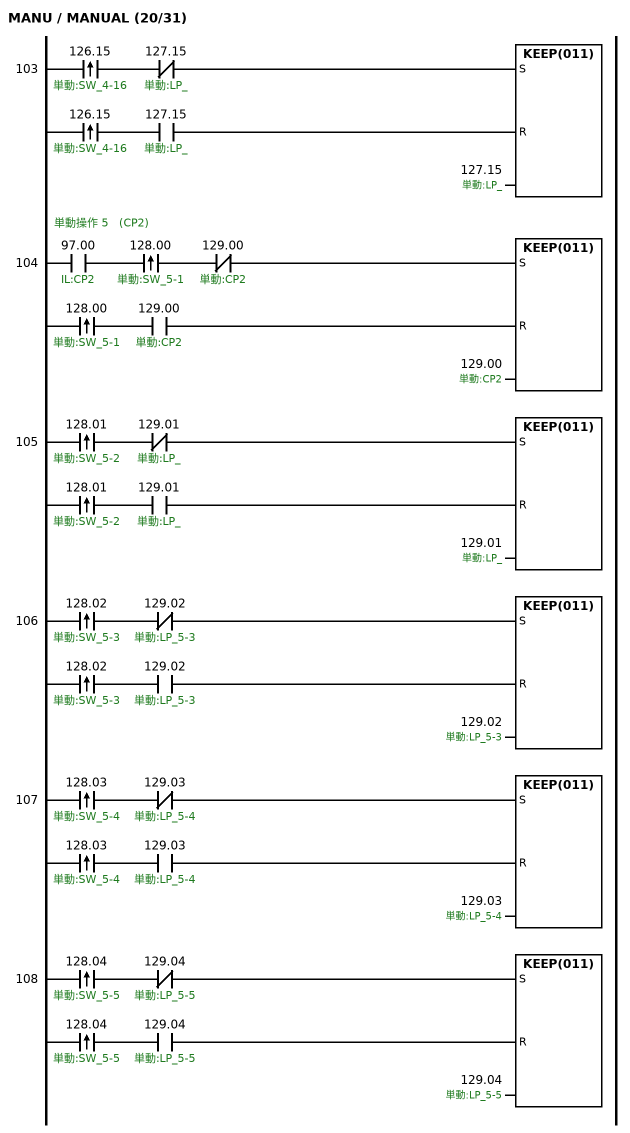
; [picture p72: MANU / MANUAL, rungs 103-108]
; rung 103
@LD 126.15  ; 単動:SW_4-16
ANDNOT 127.15  ; 単動:LP_
@LD 126.15  ; 単動:SW_4-16
AND 127.15  ; 単動:LP_
KEEP(011) 127.15  ; 単動:LP_
; rung 104: 単動操作 5   (CP2)
LD 97.00  ; IL:CP2
@AND 128.00  ; 単動:SW_5-1
ANDNOT 129.00  ; 単動:CP2
@LD 128.00  ; 単動:SW_5-1
AND 129.00  ; 単動:CP2
KEEP(011) 129.00  ; 単動:CP2
; rung 105
@LD 128.01  ; 単動:SW_5-2
ANDNOT 129.01  ; 単動:LP_
@LD 128.01  ; 単動:SW_5-2
AND 129.01  ; 単動:LP_
KEEP(011) 129.01  ; 単動:LP_
; rung 106
@LD 128.02  ; 単動:SW_5-3
ANDNOT 129.02  ; 単動:LP_5-3
@LD 128.02  ; 単動:SW_5-3
AND 129.02  ; 単動:LP_5-3
KEEP(011) 129.02  ; 単動:LP_5-3
; rung 107
@LD 128.03  ; 単動:SW_5-4
ANDNOT 129.03  ; 単動:LP_5-4
@LD 128.03  ; 単動:SW_5-4
AND 129.03  ; 単動:LP_5-4
KEEP(011) 129.03  ; 単動:LP_5-4
; rung 108
@LD 128.04  ; 単動:SW_5-5
ANDNOT 129.04  ; 単動:LP_5-5
@LD 128.04  ; 単動:SW_5-5
AND 129.04  ; 単動:LP_5-5
KEEP(011) 129.04  ; 単動:LP_5-5

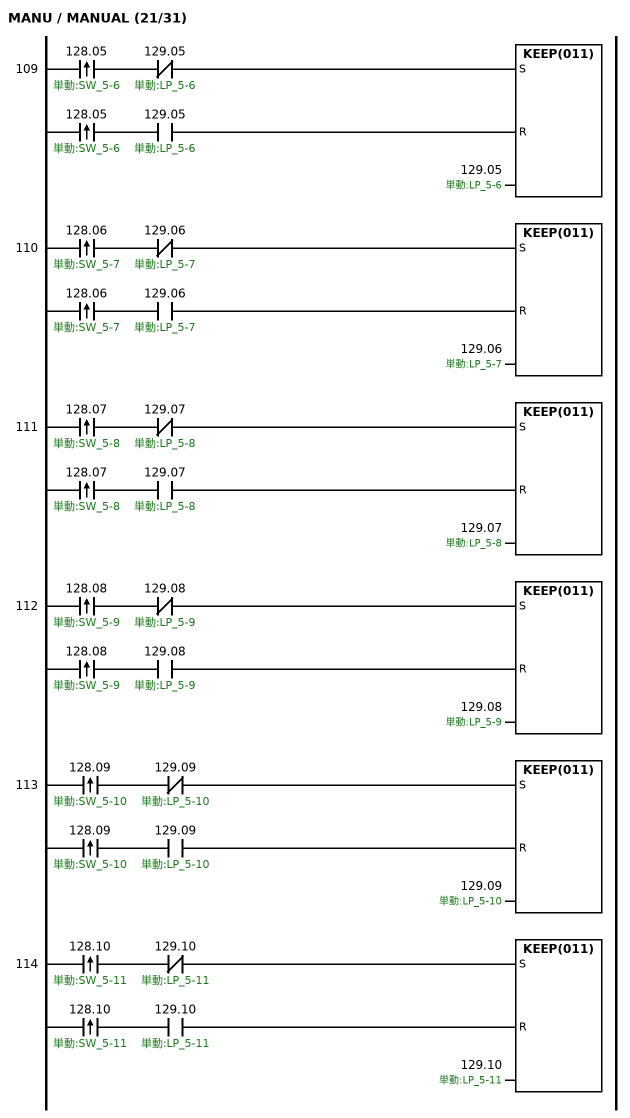
; rung 109
@LD 128.05  ; 単動:SW_5-6
ANDNOT 129.05  ; 単動:LP_5-6
@LD 128.05  ; 単動:SW_5-6
AND 129.05  ; 単動:LP_5-6
KEEP(011) 129.05  ; 単動:LP_5-6
; rung 110
@LD 128.06  ; 単動:SW_5-7
ANDNOT 129.06  ; 単動:LP_5-7
@LD 128.06  ; 単動:SW_5-7
AND 129.06  ; 単動:LP_5-7
KEEP(011) 129.06  ; 単動:LP_5-7
; rung 111
@LD 128.07  ; 単動:SW_5-8
ANDNOT 129.07  ; 単動:LP_5-8
@LD 128.07  ; 単動:SW_5-8
AND 129.07  ; 単動:LP_5-8
KEEP(011) 129.07  ; 単動:LP_5-8
; rung 112
@LD 128.08  ; 単動:SW_5-9
ANDNOT 129.08  ; 単動:LP_5-9
@LD 128.08  ; 単動:SW_5-9
AND 129.08  ; 単動:LP_5-9
KEEP(011) 129.08  ; 単動:LP_5-9
; rung 113
@LD 128.09  ; 単動:SW_5-10
ANDNOT 129.09  ; 単動:LP_5-10
@LD 128.09  ; 単動:SW_5-10
AND 129.09  ; 単動:LP_5-10
KEEP(011) 129.09  ; 単動:LP_5-10
; rung 114
@LD 128.10  ; 単動:SW_5-11
ANDNOT 129.10  ; 単動:LP_5-11
@LD 128.10  ; 単動:SW_5-11
AND 129.10  ; 単動:LP_5-11
KEEP(011) 129.10  ; 単動:LP_5-11

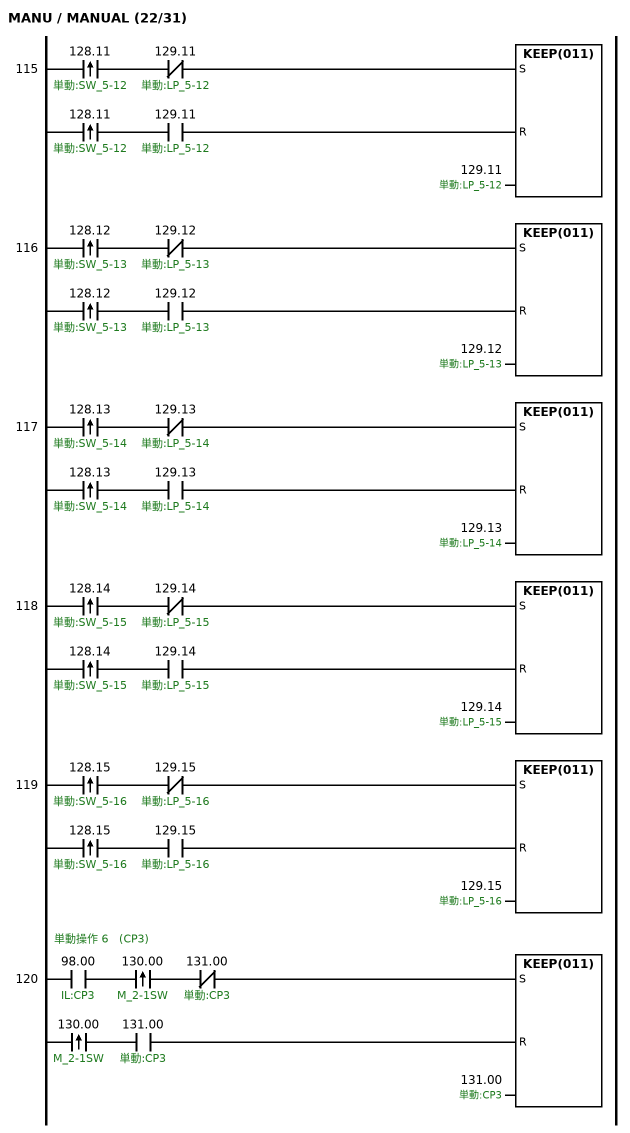
; rung 115
@LD 128.11  ; 単動:SW_5-12
ANDNOT 129.11  ; 単動:LP_5-12
@LD 128.11  ; 単動:SW_5-12
AND 129.11  ; 単動:LP_5-12
KEEP(011) 129.11  ; 単動:LP_5-12
; rung 116
@LD 128.12  ; 単動:SW_5-13
ANDNOT 129.12  ; 単動:LP_5-13
@LD 128.12  ; 単動:SW_5-13
AND 129.12  ; 単動:LP_5-13
KEEP(011) 129.12  ; 単動:LP_5-13
; rung 117
@LD 128.13  ; 単動:SW_5-14
ANDNOT 129.13  ; 単動:LP_5-14
@LD 128.13  ; 単動:SW_5-14
AND 129.13  ; 単動:LP_5-14
KEEP(011) 129.13  ; 単動:LP_5-14
; rung 118
@LD 128.14  ; 単動:SW_5-15
ANDNOT 129.14  ; 単動:LP_5-15
@LD 128.14  ; 単動:SW_5-15
AND 129.14  ; 単動:LP_5-15
KEEP(011) 129.14  ; 単動:LP_5-15
; rung 119
@LD 128.15  ; 単動:SW_5-16
ANDNOT 129.15  ; 単動:LP_5-16
@LD 128.15  ; 単動:SW_5-16
AND 129.15  ; 単動:LP_5-16
KEEP(011) 129.15  ; 単動:LP_5-16
; rung 120: 単動操作 6   (CP3)
LD 98.00  ; IL:CP3
@AND 130.00  ; M_2-1SW
ANDNOT 131.00  ; 単動:CP3
@LD 130.00  ; M_2-1SW
AND 131.00  ; 単動:CP3
KEEP(011) 131.00  ; 単動:CP3

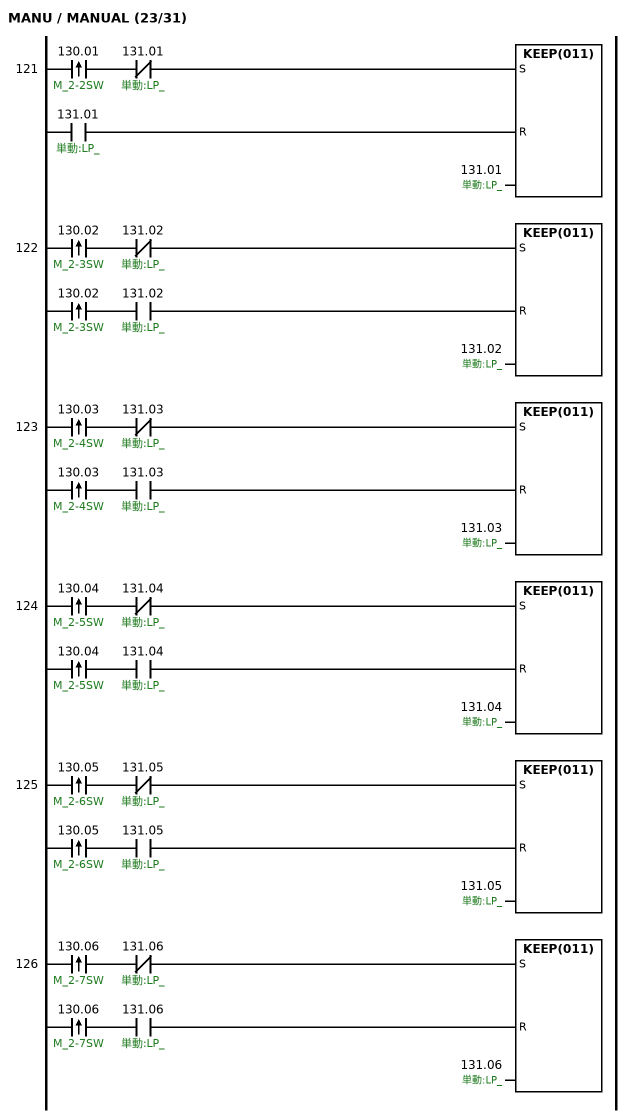
; rung 121
@LD 130.01  ; M_2-2SW
ANDNOT 131.01  ; 単動:LP_
LD 131.01  ; 単動:LP_
KEEP(011) 131.01  ; 単動:LP_
; rung 122
@LD 130.02  ; M_2-3SW
ANDNOT 131.02  ; 単動:LP_
@LD 130.02  ; M_2-3SW
AND 131.02  ; 単動:LP_
KEEP(011) 131.02  ; 単動:LP_
; rung 123
@LD 130.03  ; M_2-4SW
ANDNOT 131.03  ; 単動:LP_
@LD 130.03  ; M_2-4SW
AND 131.03  ; 単動:LP_
KEEP(011) 131.03  ; 単動:LP_
; rung 124
@LD 130.04  ; M_2-5SW
ANDNOT 131.04  ; 単動:LP_
@LD 130.04  ; M_2-5SW
AND 131.04  ; 単動:LP_
KEEP(011) 131.04  ; 単動:LP_
; rung 125
@LD 130.05  ; M_2-6SW
ANDNOT 131.05  ; 単動:LP_
@LD 130.05  ; M_2-6SW
AND 131.05  ; 単動:LP_
KEEP(011) 131.05  ; 単動:LP_
; rung 126
@LD 130.06  ; M_2-7SW
ANDNOT 131.06  ; 単動:LP_
@LD 130.06  ; M_2-7SW
AND 131.06  ; 単動:LP_
KEEP(011) 131.06  ; 単動:LP_

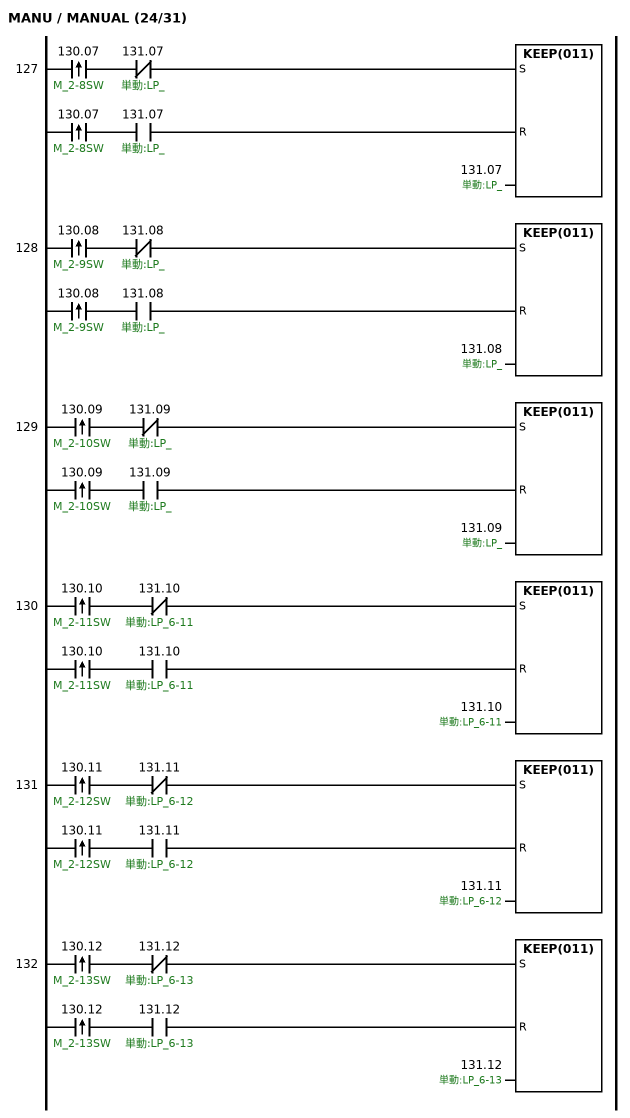
; rung 127
@LD 130.07  ; M_2-8SW
ANDNOT 131.07  ; 単動:LP_
@LD 130.07  ; M_2-8SW
AND 131.07  ; 単動:LP_
KEEP(011) 131.07  ; 単動:LP_
; rung 128
@LD 130.08  ; M_2-9SW
ANDNOT 131.08  ; 単動:LP_
@LD 130.08  ; M_2-9SW
AND 131.08  ; 単動:LP_
KEEP(011) 131.08  ; 単動:LP_
; rung 129
@LD 130.09  ; M_2-10SW
ANDNOT 131.09  ; 単動:LP_
@LD 130.09  ; M_2-10SW
AND 131.09  ; 単動:LP_
KEEP(011) 131.09  ; 単動:LP_
; rung 130
@LD 130.10  ; M_2-11SW
ANDNOT 131.10  ; 単動:LP_6-11
@LD 130.10  ; M_2-11SW
AND 131.10  ; 単動:LP_6-11
KEEP(011) 131.10  ; 単動:LP_6-11
; rung 131
@LD 130.11  ; M_2-12SW
ANDNOT 131.11  ; 単動:LP_6-12
@LD 130.11  ; M_2-12SW
AND 131.11  ; 単動:LP_6-12
KEEP(011) 131.11  ; 単動:LP_6-12
; rung 132
@LD 130.12  ; M_2-13SW
ANDNOT 131.12  ; 単動:LP_6-13
@LD 130.12  ; M_2-13SW
AND 131.12  ; 単動:LP_6-13
KEEP(011) 131.12  ; 単動:LP_6-13

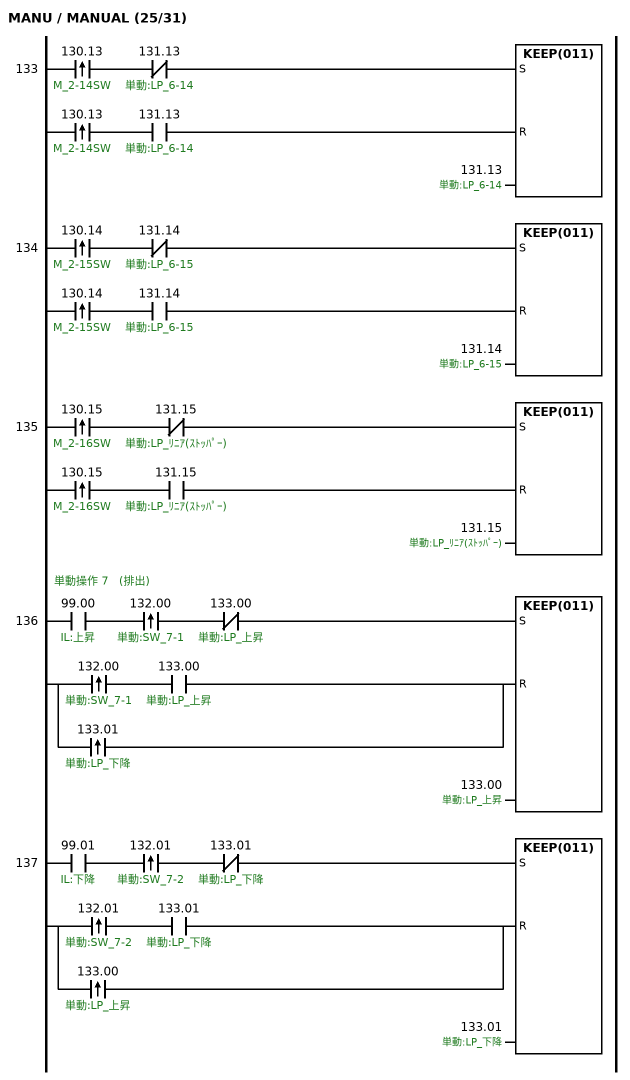
; rung 133
@LD 130.13  ; M_2-14SW
ANDNOT 131.13  ; 単動:LP_6-14
@LD 130.13  ; M_2-14SW
AND 131.13  ; 単動:LP_6-14
KEEP(011) 131.13  ; 単動:LP_6-14
; rung 134
@LD 130.14  ; M_2-15SW
ANDNOT 131.14  ; 単動:LP_6-15
@LD 130.14  ; M_2-15SW
AND 131.14  ; 単動:LP_6-15
KEEP(011) 131.14  ; 単動:LP_6-15
; rung 135
@LD 130.15  ; M_2-16SW
ANDNOT 131.15  ; 単動:LP_ﾘﾆｱ(ｽﾄｯﾊﾟｰ)
@LD 130.15  ; M_2-16SW
AND 131.15  ; 単動:LP_ﾘﾆｱ(ｽﾄｯﾊﾟｰ)
KEEP(011) 131.15  ; 単動:LP_ﾘﾆｱ(ｽﾄｯﾊﾟｰ)
; rung 136: 単動操作 7   (排出)
LD 99.00  ; IL:上昇
@AND 132.00  ; 単動:SW_7-1
ANDNOT 133.00  ; 単動:LP_上昇
@LD 132.00  ; 単動:SW_7-1
AND 133.00  ; 単動:LP_上昇
@OR 133.01  ; 単動:LP_下降
KEEP(011) 133.00  ; 単動:LP_上昇
; rung 137
LD 99.01  ; IL:下降
@AND 132.01  ; 単動:SW_7-2
ANDNOT 133.01  ; 単動:LP_下降
@LD 132.01  ; 単動:SW_7-2
AND 133.01  ; 単動:LP_下降
@OR 133.00  ; 単動:LP_上昇
KEEP(011) 133.01  ; 単動:LP_下降

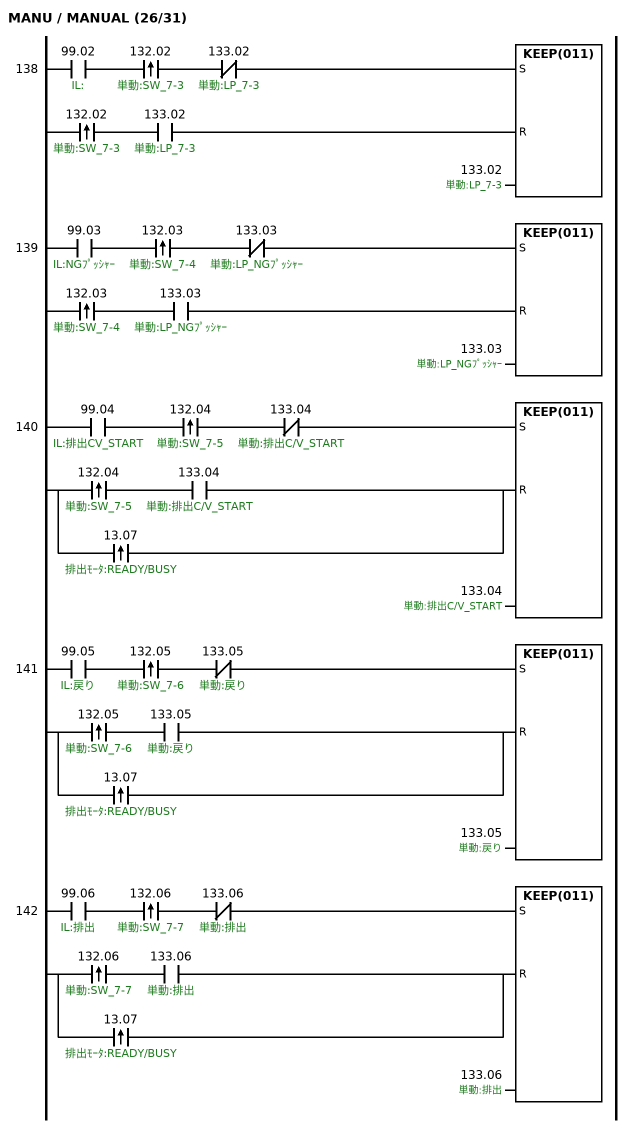
; rung 138
LD 99.02  ; IL:
@AND 132.02  ; 単動:SW_7-3
ANDNOT 133.02  ; 単動:LP_7-3
@LD 132.02  ; 単動:SW_7-3
AND 133.02  ; 単動:LP_7-3
KEEP(011) 133.02  ; 単動:LP_7-3
; rung 139
LD 99.03  ; IL:NGﾌﾟｯｼｬｰ
@AND 132.03  ; 単動:SW_7-4
ANDNOT 133.03  ; 単動:LP_NGﾌﾟｯｼｬｰ
@LD 132.03  ; 単動:SW_7-4
AND 133.03  ; 単動:LP_NGﾌﾟｯｼｬｰ
KEEP(011) 133.03  ; 単動:LP_NGﾌﾟｯｼｬｰ
; rung 140
LD 99.04  ; IL:排出CV_START
@AND 132.04  ; 単動:SW_7-5
ANDNOT 133.04  ; 単動:排出C/V_START
@LD 132.04  ; 単動:SW_7-5
AND 133.04  ; 単動:排出C/V_START
@OR 13.07  ; 排出ﾓｰﾀ:READY/BUSY
KEEP(011) 133.04  ; 単動:排出C/V_START
; rung 141
LD 99.05  ; IL:戻り
@AND 132.05  ; 単動:SW_7-6
ANDNOT 133.05  ; 単動:戻り
@LD 132.05  ; 単動:SW_7-6
AND 133.05  ; 単動:戻り
@OR 13.07  ; 排出ﾓｰﾀ:READY/BUSY
KEEP(011) 133.05  ; 単動:戻り
; rung 142
LD 99.06  ; IL:排出
@AND 132.06  ; 単動:SW_7-7
ANDNOT 133.06  ; 単動:排出
@LD 132.06  ; 単動:SW_7-7
AND 133.06  ; 単動:排出
@OR 13.07  ; 排出ﾓｰﾀ:READY/BUSY
KEEP(011) 133.06  ; 単動:排出

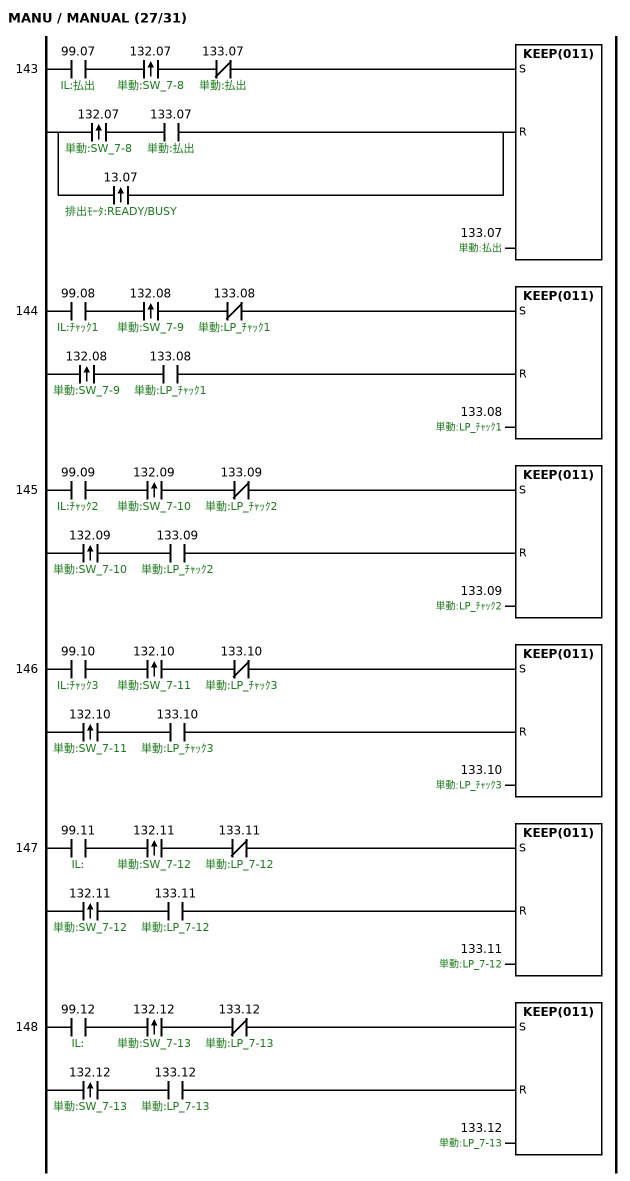
; rung 143
LD 99.07  ; IL:払出
@AND 132.07  ; 単動:SW_7-8
ANDNOT 133.07  ; 単動:払出
@LD 132.07  ; 単動:SW_7-8
AND 133.07  ; 単動:払出
@OR 13.07  ; 排出ﾓｰﾀ:READY/BUSY
KEEP(011) 133.07  ; 単動:払出
; rung 144
LD 99.08  ; IL:ﾁｬｯｸ1
@AND 132.08  ; 単動:SW_7-9
ANDNOT 133.08  ; 単動:LP_ﾁｬｯｸ1
@LD 132.08  ; 単動:SW_7-9
AND 133.08  ; 単動:LP_ﾁｬｯｸ1
KEEP(011) 133.08  ; 単動:LP_ﾁｬｯｸ1
; rung 145
LD 99.09  ; IL:ﾁｬｯｸ2
@AND 132.09  ; 単動:SW_7-10
ANDNOT 133.09  ; 単動:LP_ﾁｬｯｸ2
@LD 132.09  ; 単動:SW_7-10
AND 133.09  ; 単動:LP_ﾁｬｯｸ2
KEEP(011) 133.09  ; 単動:LP_ﾁｬｯｸ2
; rung 146
LD 99.10  ; IL:ﾁｬｯｸ3
@AND 132.10  ; 単動:SW_7-11
ANDNOT 133.10  ; 単動:LP_ﾁｬｯｸ3
@LD 132.10  ; 単動:SW_7-11
AND 133.10  ; 単動:LP_ﾁｬｯｸ3
KEEP(011) 133.10  ; 単動:LP_ﾁｬｯｸ3
; rung 147
LD 99.11  ; IL:
@AND 132.11  ; 単動:SW_7-12
ANDNOT 133.11  ; 単動:LP_7-12
@LD 132.11  ; 単動:SW_7-12
AND 133.11  ; 単動:LP_7-12
KEEP(011) 133.11  ; 単動:LP_7-12
; rung 148
LD 99.12  ; IL:
@AND 132.12  ; 単動:SW_7-13
ANDNOT 133.12  ; 単動:LP_7-13
@LD 132.12  ; 単動:SW_7-13
AND 133.12  ; 単動:LP_7-13
KEEP(011) 133.12  ; 単動:LP_7-13

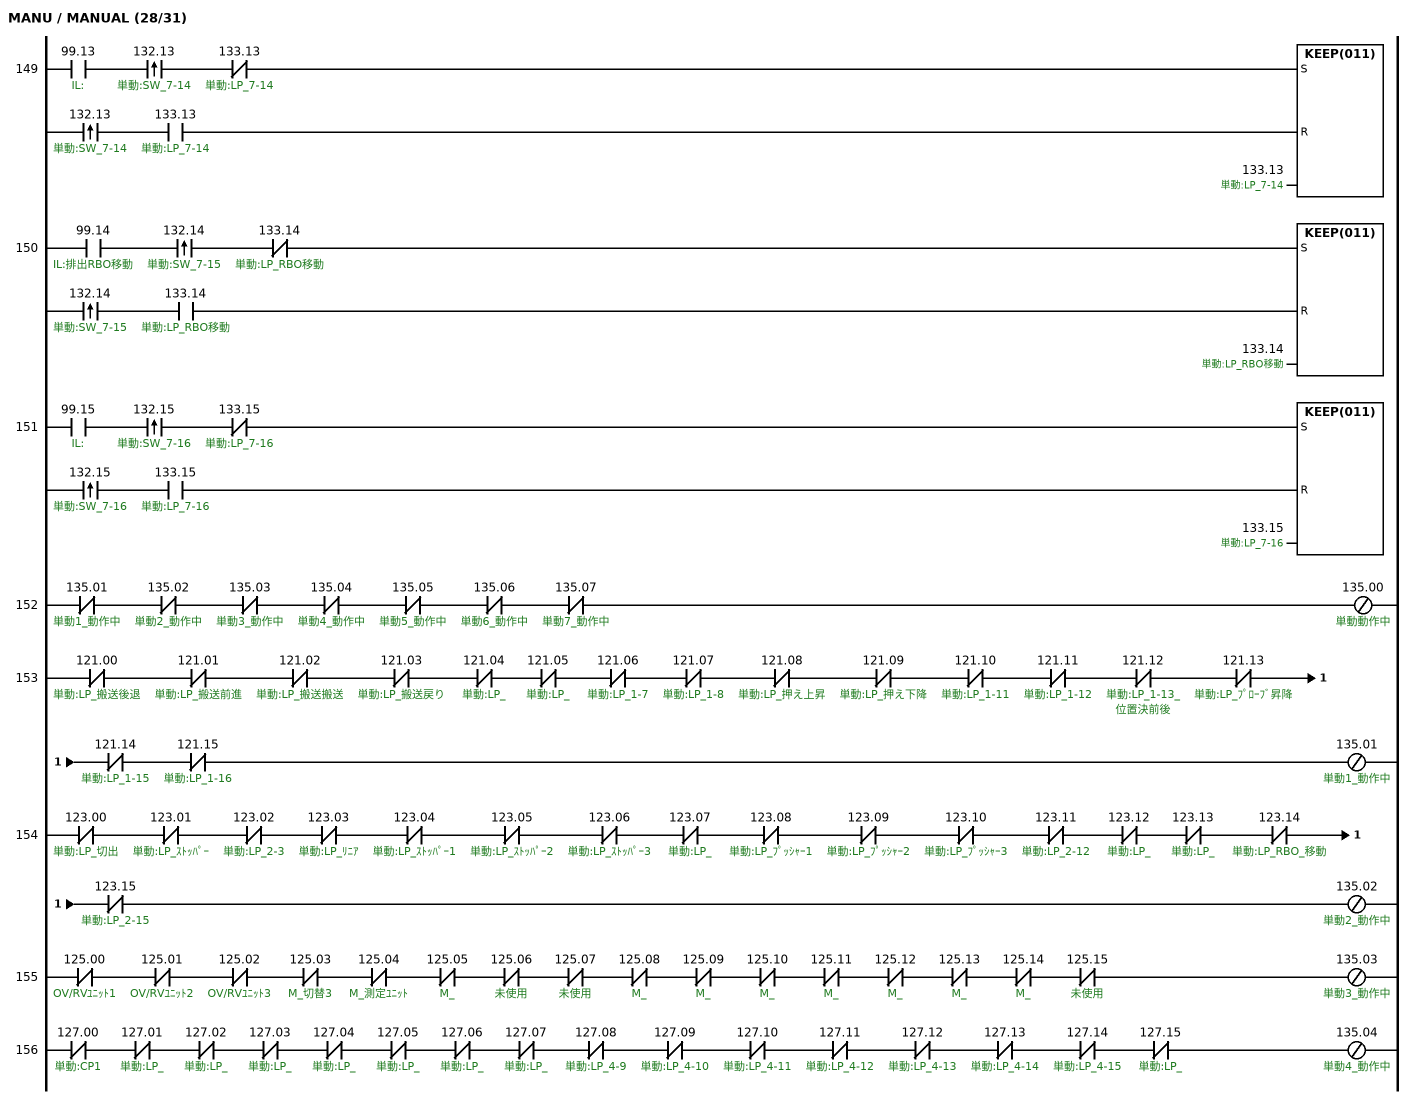
; rung 149
LD 99.13  ; IL:
@AND 132.13  ; 単動:SW_7-14
ANDNOT 133.13  ; 単動:LP_7-14
@LD 132.13  ; 単動:SW_7-14
AND 133.13  ; 単動:LP_7-14
KEEP(011) 133.13  ; 単動:LP_7-14
; rung 150
LD 99.14  ; IL:排出RBO移動
@AND 132.14  ; 単動:SW_7-15
ANDNOT 133.14  ; 単動:LP_RBO移動
@LD 132.14  ; 単動:SW_7-15
AND 133.14  ; 単動:LP_RBO移動
KEEP(011) 133.14  ; 単動:LP_RBO移動
; rung 151
LD 99.15  ; IL:
@AND 132.15  ; 単動:SW_7-16
ANDNOT 133.15  ; 単動:LP_7-16
@LD 132.15  ; 単動:SW_7-16
AND 133.15  ; 単動:LP_7-16
KEEP(011) 133.15  ; 単動:LP_7-16
; rung 152
LDNOT 135.01  ; 単動1_動作中
ANDNOT 135.02  ; 単動2_動作中
ANDNOT 135.03  ; 単動3_動作中
ANDNOT 135.04  ; 単動4_動作中
ANDNOT 135.05  ; 単動5_動作中
ANDNOT 135.06  ; 単動6_動作中
ANDNOT 135.07  ; 単動7_動作中
OUTNOT 135.00  ; 単動動作中
; rung 153
LDNOT 121.00  ; 単動:LP_搬送後退
ANDNOT 121.01  ; 単動:LP_搬送前進
ANDNOT 121.02  ; 単動:LP_搬送搬送
ANDNOT 121.03  ; 単動:LP_搬送戻り
ANDNOT 121.04  ; 単動:LP_
ANDNOT 121.05  ; 単動:LP_
ANDNOT 121.06  ; 単動:LP_1-7
ANDNOT 121.07  ; 単動:LP_1-8
ANDNOT 121.08  ; 単動:LP_押え上昇
ANDNOT 121.09  ; 単動:LP_押え下降
ANDNOT 121.10  ; 単動:LP_1-11
ANDNOT 121.11  ; 単動:LP_1-12
ANDNOT 121.12  ; 単動:LP_1-13_位置決前後
ANDNOT 121.13  ; 単動:LP_ﾌﾟﾛｰﾌﾞ昇降
ANDNOT 121.14  ; 単動:LP_1-15
ANDNOT 121.15  ; 単動:LP_1-16
OUTNOT 135.01  ; 単動1_動作中
; rung 154
LDNOT 123.00  ; 単動:LP_切出
ANDNOT 123.01  ; 単動:LP_ｽﾄｯﾊﾟｰ
ANDNOT 123.02  ; 単動:LP_2-3
ANDNOT 123.03  ; 単動:LP_ﾘﾆｱ
ANDNOT 123.04  ; 単動:LP_ｽﾄｯﾊﾟｰ1
ANDNOT 123.05  ; 単動:LP_ｽﾄｯﾊﾟｰ2
ANDNOT 123.06  ; 単動:LP_ｽﾄｯﾊﾟｰ3
ANDNOT 123.07  ; 単動:LP_
ANDNOT 123.08  ; 単動:LP_ﾌﾟｯｼｬｰ1
ANDNOT 123.09  ; 単動:LP_ﾌﾟｯｼｬｰ2
ANDNOT 123.10  ; 単動:LP_ﾌﾟｯｼｬｰ3
ANDNOT 123.11  ; 単動:LP_2-12
ANDNOT 123.12  ; 単動:LP_
ANDNOT 123.13  ; 単動:LP_
ANDNOT 123.14  ; 単動:LP_RBO_移動
ANDNOT 123.15  ; 単動:LP_2-15
OUTNOT 135.02  ; 単動2_動作中
; rung 155
LDNOT 125.00  ; OV/RVﾕﾆｯﾄ1
ANDNOT 125.01  ; OV/RVﾕﾆｯﾄ2
ANDNOT 125.02  ; OV/RVﾕﾆｯﾄ3
ANDNOT 125.03  ; M_切替3
ANDNOT 125.04  ; M_測定ﾕﾆｯﾄ
ANDNOT 125.05  ; M_
ANDNOT 125.06  ; 未使用
ANDNOT 125.07  ; 未使用
ANDNOT 125.08  ; M_
ANDNOT 125.09  ; M_
ANDNOT 125.10  ; M_
ANDNOT 125.11  ; M_
ANDNOT 125.12  ; M_
ANDNOT 125.13  ; M_
ANDNOT 125.14  ; M_
ANDNOT 125.15  ; 未使用
OUTNOT 135.03  ; 単動3_動作中
; rung 156
LDNOT 127.00  ; 単動:CP1
ANDNOT 127.01  ; 単動:LP_
ANDNOT 127.02  ; 単動:LP_
ANDNOT 127.03  ; 単動:LP_
ANDNOT 127.04  ; 単動:LP_
ANDNOT 127.05  ; 単動:LP_
ANDNOT 127.06  ; 単動:LP_
ANDNOT 127.07  ; 単動:LP_
ANDNOT 127.08  ; 単動:LP_4-9
ANDNOT 127.09  ; 単動:LP_4-10
ANDNOT 127.10  ; 単動:LP_4-11
ANDNOT 127.11  ; 単動:LP_4-12
ANDNOT 127.12  ; 単動:LP_4-13
ANDNOT 127.13  ; 単動:LP_4-14
ANDNOT 127.14  ; 単動:LP_4-15
ANDNOT 127.15  ; 単動:LP_
OUTNOT 135.04  ; 単動4_動作中

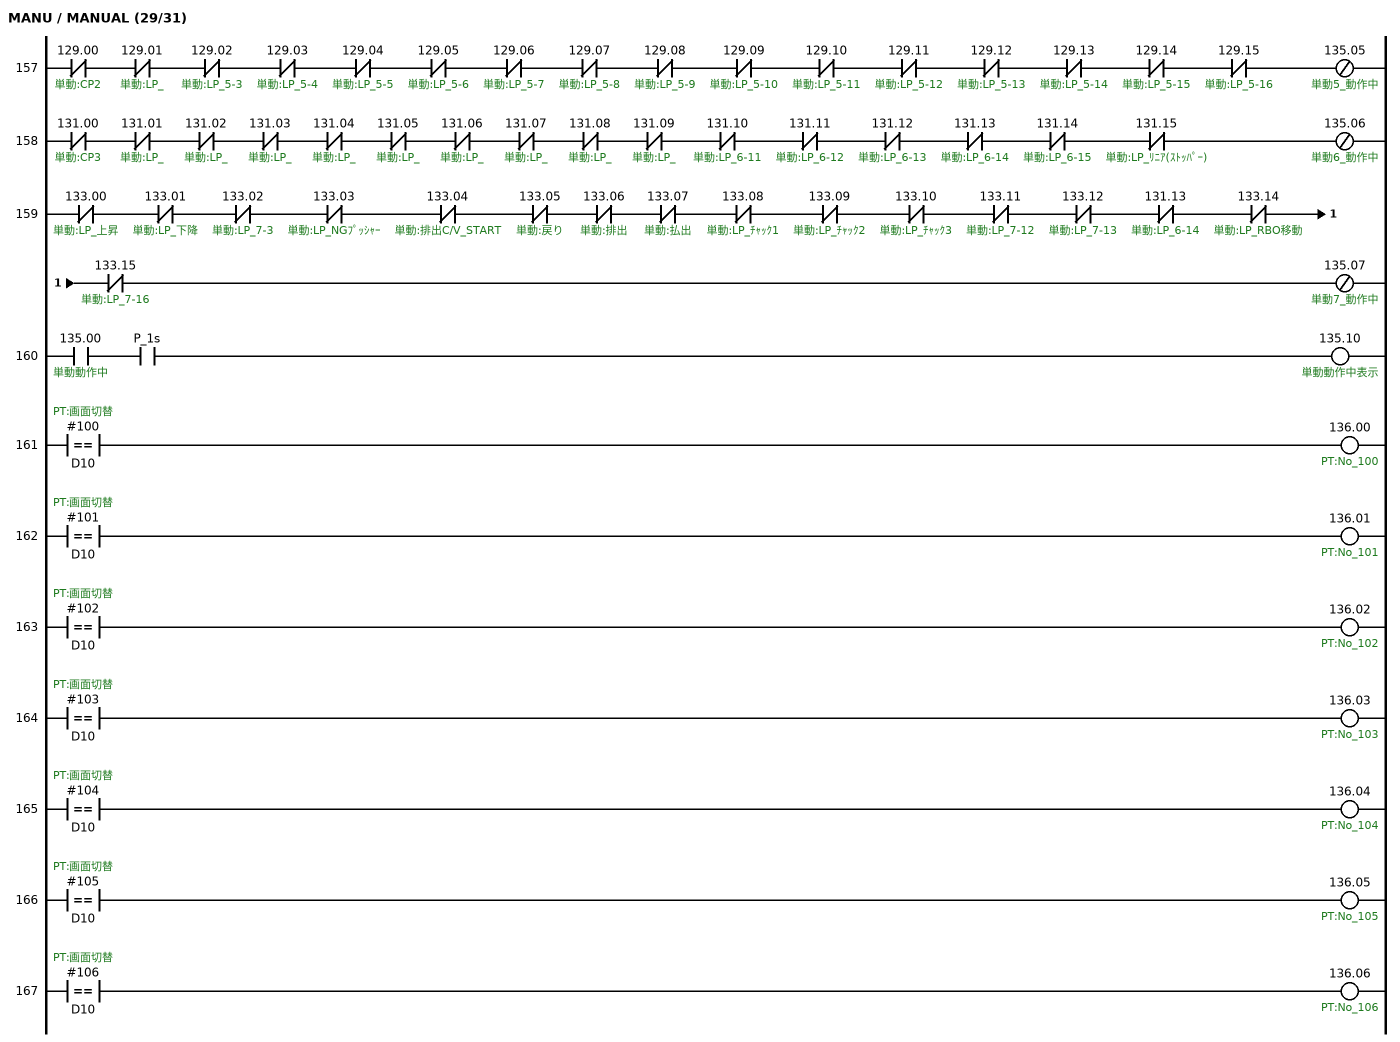
; rung 157
LDNOT 129.00  ; 単動:CP2
ANDNOT 129.01  ; 単動:LP_
ANDNOT 129.02  ; 単動:LP_5-3
ANDNOT 129.03  ; 単動:LP_5-4
ANDNOT 129.04  ; 単動:LP_5-5
ANDNOT 129.05  ; 単動:LP_5-6
ANDNOT 129.06  ; 単動:LP_5-7
ANDNOT 129.07  ; 単動:LP_5-8
ANDNOT 129.08  ; 単動:LP_5-9
ANDNOT 129.09  ; 単動:LP_5-10
ANDNOT 129.10  ; 単動:LP_5-11
ANDNOT 129.11  ; 単動:LP_5-12
ANDNOT 129.12  ; 単動:LP_5-13
ANDNOT 129.13  ; 単動:LP_5-14
ANDNOT 129.14  ; 単動:LP_5-15
ANDNOT 129.15  ; 単動:LP_5-16
OUTNOT 135.05  ; 単動5_動作中
; rung 158
LDNOT 131.00  ; 単動:CP3
ANDNOT 131.01  ; 単動:LP_
ANDNOT 131.02  ; 単動:LP_
ANDNOT 131.03  ; 単動:LP_
ANDNOT 131.04  ; 単動:LP_
ANDNOT 131.05  ; 単動:LP_
ANDNOT 131.06  ; 単動:LP_
ANDNOT 131.07  ; 単動:LP_
ANDNOT 131.08  ; 単動:LP_
ANDNOT 131.09  ; 単動:LP_
ANDNOT 131.10  ; 単動:LP_6-11
ANDNOT 131.11  ; 単動:LP_6-12
ANDNOT 131.12  ; 単動:LP_6-13
ANDNOT 131.13  ; 単動:LP_6-14
ANDNOT 131.14  ; 単動:LP_6-15
ANDNOT 131.15  ; 単動:LP_ﾘﾆｱ(ｽﾄｯﾊﾟｰ)
OUTNOT 135.06  ; 単動6_動作中
; rung 159
LDNOT 133.00  ; 単動:LP_上昇
ANDNOT 133.01  ; 単動:LP_下降
ANDNOT 133.02  ; 単動:LP_7-3
ANDNOT 133.03  ; 単動:LP_NGﾌﾟｯｼｬｰ
ANDNOT 133.04  ; 単動:排出C/V_START
ANDNOT 133.05  ; 単動:戻り
ANDNOT 133.06  ; 単動:排出
ANDNOT 133.07  ; 単動:払出
ANDNOT 133.08  ; 単動:LP_ﾁｬｯｸ1
ANDNOT 133.09  ; 単動:LP_ﾁｬｯｸ2
ANDNOT 133.10  ; 単動:LP_ﾁｬｯｸ3
ANDNOT 133.11  ; 単動:LP_7-12
ANDNOT 133.12  ; 単動:LP_7-13
ANDNOT 131.13  ; 単動:LP_6-14
ANDNOT 133.14  ; 単動:LP_RBO移動
ANDNOT 133.15  ; 単動:LP_7-16
OUTNOT 135.07  ; 単動7_動作中
; rung 160
LD 135.00  ; 単動動作中
AND P_1s
OUT 135.10  ; 単動動作中表示
; rung 161
LD=(300) #100 D10  ; PT:画面切替
OUT 136.00  ; PT:No_100
; rung 162
LD=(300) #101 D10  ; PT:画面切替
OUT 136.01  ; PT:No_101
; rung 163
LD=(300) #102 D10  ; PT:画面切替
OUT 136.02  ; PT:No_102
; rung 164
LD=(300) #103 D10  ; PT:画面切替
OUT 136.03  ; PT:No_103
; rung 165
LD=(300) #104 D10  ; PT:画面切替
OUT 136.04  ; PT:No_104
; rung 166
LD=(300) #105 D10  ; PT:画面切替
OUT 136.05  ; PT:No_105
; rung 167
LD=(300) #106 D10  ; PT:画面切替
OUT 136.06  ; PT:No_106

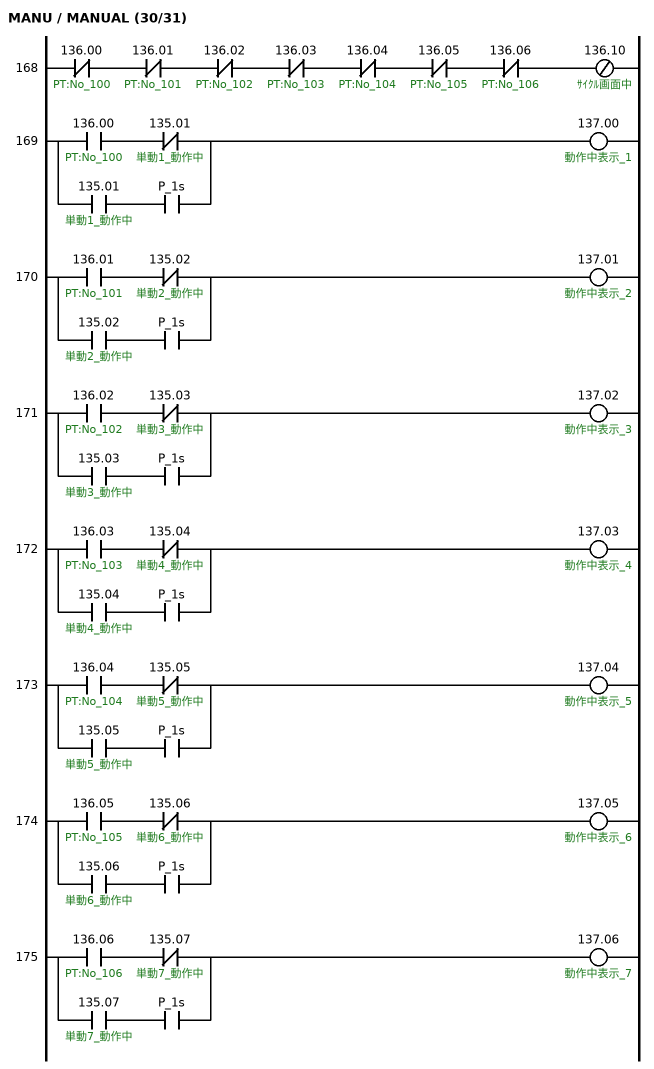
; rung 168
LDNOT 136.00  ; PT:No_100
ANDNOT 136.01  ; PT:No_101
ANDNOT 136.02  ; PT:No_102
ANDNOT 136.03  ; PT:No_103
ANDNOT 136.04  ; PT:No_104
ANDNOT 136.05  ; PT:No_105
ANDNOT 136.06  ; PT:No_106
OUTNOT 136.10  ; ｻｲｸﾙ画面中
; rung 169
LD 136.00  ; PT:No_100
ANDNOT 135.01  ; 単動1_動作中
LD 135.01  ; 単動1_動作中
AND P_1s
ORLD
OUT 137.00  ; 動作中表示_1
; rung 170
LD 136.01  ; PT:No_101
ANDNOT 135.02  ; 単動2_動作中
LD 135.02  ; 単動2_動作中
AND P_1s
ORLD
OUT 137.01  ; 動作中表示_2
; rung 171
LD 136.02  ; PT:No_102
ANDNOT 135.03  ; 単動3_動作中
LD 135.03  ; 単動3_動作中
AND P_1s
ORLD
OUT 137.02  ; 動作中表示_3
; rung 172
LD 136.03  ; PT:No_103
ANDNOT 135.04  ; 単動4_動作中
LD 135.04  ; 単動4_動作中
AND P_1s
ORLD
OUT 137.03  ; 動作中表示_4
; rung 173
LD 136.04  ; PT:No_104
ANDNOT 135.05  ; 単動5_動作中
LD 135.05  ; 単動5_動作中
AND P_1s
ORLD
OUT 137.04  ; 動作中表示_5
; rung 174
LD 136.05  ; PT:No_105
ANDNOT 135.06  ; 単動6_動作中
LD 135.06  ; 単動6_動作中
AND P_1s
ORLD
OUT 137.05  ; 動作中表示_6
; rung 175
LD 136.06  ; PT:No_106
ANDNOT 135.07  ; 単動7_動作中
LD 135.07  ; 単動7_動作中
AND P_1s
ORLD
OUT 137.06  ; 動作中表示_7

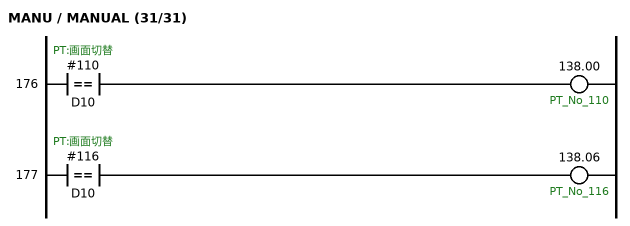
; rung 176
LD=(300) #110 D10  ; PT:画面切替
OUT 138.00  ; PT_No_110
; rung 177
LD=(300) #116 D10  ; PT:画面切替
OUT 138.06  ; PT_No_116

### Section END
; rung 0
END(001)

## Program 主軸 (cyclic task 2)

### Section 動作制御

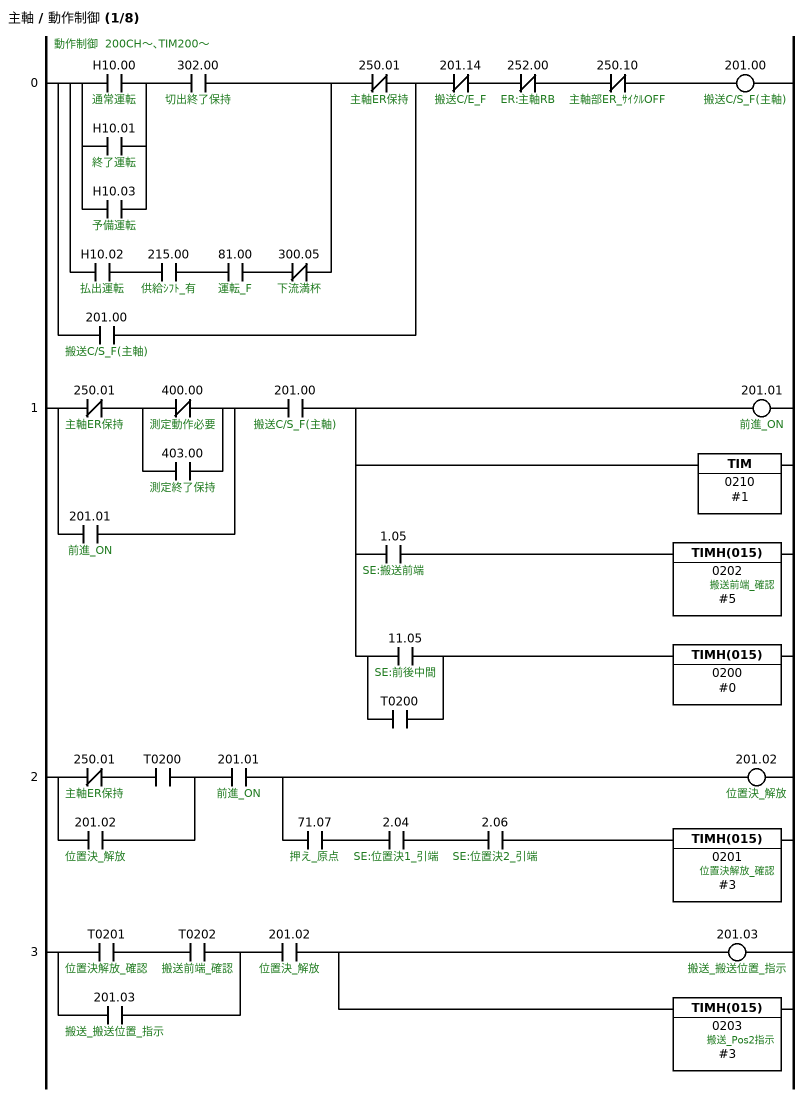
; rung 0: 動作制御  200CH～､TIM200～
LD H10.00  ; 通常運転
OR H10.01  ; 終了運転
OR H10.03  ; 予備運転
AND 302.00  ; 切出終了保持
LD H10.02  ; 払出運転
AND 215.00  ; 供給ｼﾌﾄ_有
AND 81.00  ; 運転_F
ANDNOT 300.05  ; 下流満杯
ORLD
ANDNOT 250.01  ; 主軸ER保持
OR 201.00  ; 搬送C/S_F(主軸)
ANDNOT 201.14  ; 搬送C/E_F
ANDNOT 252.00  ; ER:主軸RB
ANDNOT 250.10  ; 主軸部ER_ｻｲｸﾙOFF
OUT 201.00  ; 搬送C/S_F(主軸)
; rung 1
LDNOT 250.01  ; 主軸ER保持
LDNOT 400.00  ; 測定動作必要
OR 403.00  ; 測定終了保持
ANDLD
OR 201.01  ; 前進_ON
AND 201.00  ; 搬送C/S_F(主軸)
OUT TR0
OUT 201.01  ; 前進_ON
TIM 0210 #1
AND 1.05  ; SE:搬送前端
TIMH(015) 0202 #5  ; 搬送前端_確認
LD TR0
LD 11.05  ; SE:前後中間
OR T0200
ANDLD
TIMH(015) 0200 #0
; rung 2
LDNOT 250.01  ; 主軸ER保持
AND T0200
OR 201.02  ; 位置決_解放
AND 201.01  ; 前進_ON
OUT 201.02  ; 位置決_解放
AND 71.07  ; 押え_原点
AND 2.04  ; SE:位置決1_引端
AND 2.06  ; SE:位置決2_引端
TIMH(015) 0201 #3  ; 位置決解放_確認
; rung 3
LD T0201  ; 位置決解放_確認
AND T0202  ; 搬送前端_確認
OR 201.03  ; 搬送_搬送位置_指示
AND 201.02  ; 位置決_解放
OUT 201.03  ; 搬送_搬送位置_指示
TIMH(015) 0203 #3  ; 搬送_Pos2指示

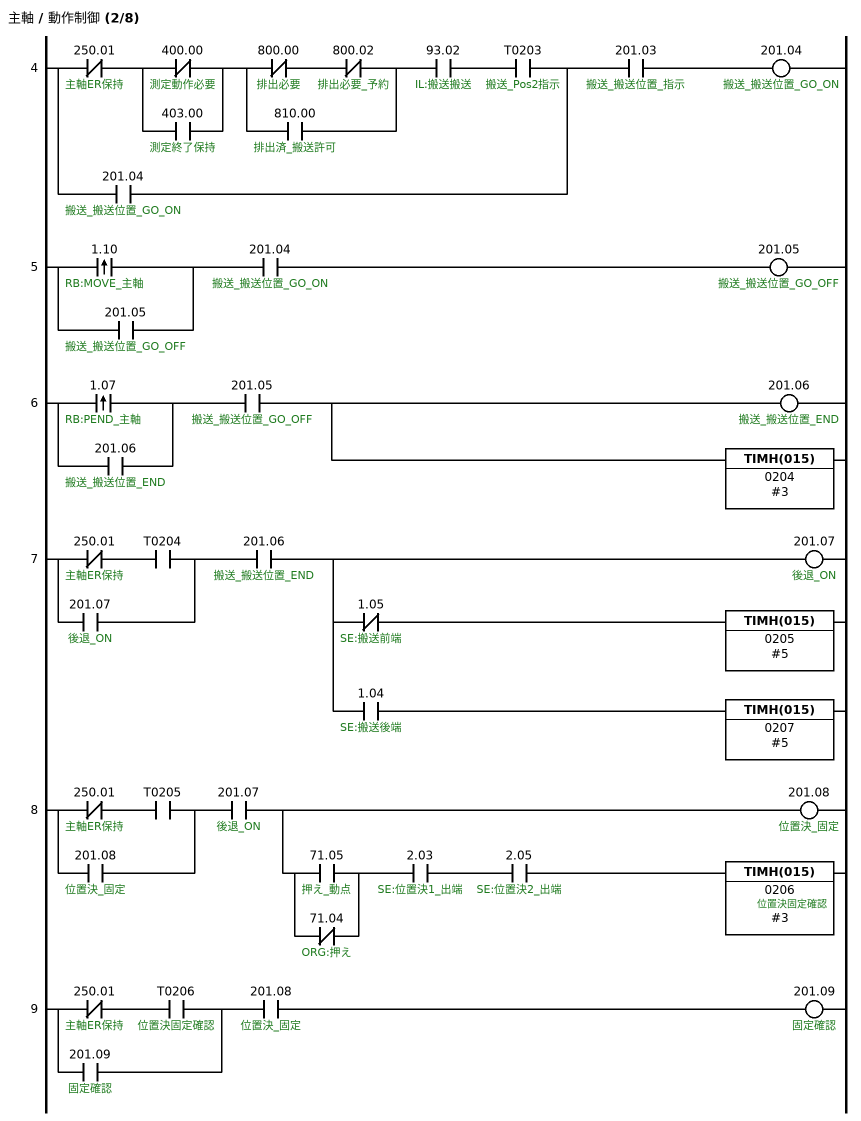
; rung 4
LDNOT 250.01  ; 主軸ER保持
LDNOT 400.00  ; 測定動作必要
OR 403.00  ; 測定終了保持
ANDLD
LDNOT 800.00  ; 排出必要
ANDNOT 800.02  ; 排出必要_予約
OR 810.00  ; 排出済_搬送許可
ANDLD
AND 93.02  ; IL:搬送搬送
AND T0203  ; 搬送_Pos2指示
OR 201.04  ; 搬送_搬送位置_GO_ON
AND 201.03  ; 搬送_搬送位置_指示
OUT 201.04  ; 搬送_搬送位置_GO_ON
; rung 5
@LD 1.10  ; RB:MOVE_主軸
OR 201.05  ; 搬送_搬送位置_GO_OFF
AND 201.04  ; 搬送_搬送位置_GO_ON
OUT 201.05  ; 搬送_搬送位置_GO_OFF
; rung 6
@LD 1.07  ; RB:PEND_主軸
OR 201.06  ; 搬送_搬送位置_END
AND 201.05  ; 搬送_搬送位置_GO_OFF
OUT 201.06  ; 搬送_搬送位置_END
TIMH(015) 0204 #3
; rung 7
LDNOT 250.01  ; 主軸ER保持
AND T0204
OR 201.07  ; 後退_ON
AND 201.06  ; 搬送_搬送位置_END
OUT TR0
OUT 201.07  ; 後退_ON
ANDNOT 1.05  ; SE:搬送前端
TIMH(015) 0205 #5
LD TR0
AND 1.04  ; SE:搬送後端
TIMH(015) 0207 #5
; rung 8
LDNOT 250.01  ; 主軸ER保持
AND T0205
OR 201.08  ; 位置決_固定
AND 201.07  ; 後退_ON
OUT 201.08  ; 位置決_固定
LD 71.05  ; 押え_動点
ORNOT 71.04  ; ORG:押え
ANDLD
AND 2.03  ; SE:位置決1_出端
AND 2.05  ; SE:位置決2_出端
TIMH(015) 0206 #3  ; 位置決固定確認
; rung 9
LDNOT 250.01  ; 主軸ER保持
AND T0206  ; 位置決固定確認
OR 201.09  ; 固定確認
AND 201.08  ; 位置決_固定
OUT 201.09  ; 固定確認

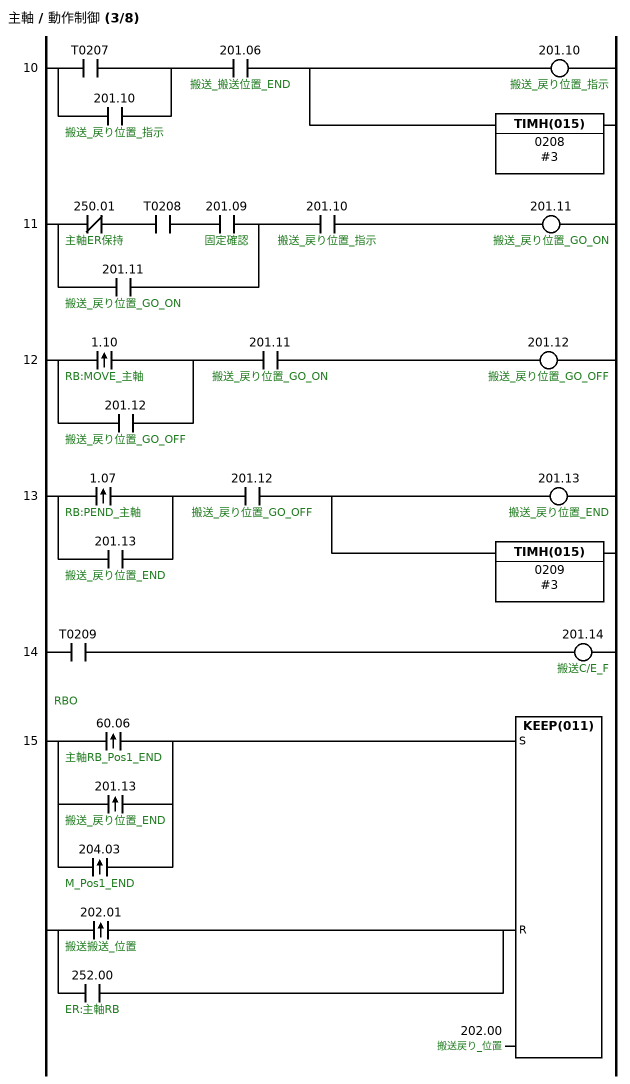
; rung 10
LD T0207
OR 201.10  ; 搬送_戻り位置_指示
AND 201.06  ; 搬送_搬送位置_END
OUT 201.10  ; 搬送_戻り位置_指示
TIMH(015) 0208 #3
; rung 11
LDNOT 250.01  ; 主軸ER保持
AND T0208
AND 201.09  ; 固定確認
OR 201.11  ; 搬送_戻り位置_GO_ON
AND 201.10  ; 搬送_戻り位置_指示
OUT 201.11  ; 搬送_戻り位置_GO_ON
; rung 12
@LD 1.10  ; RB:MOVE_主軸
OR 201.12  ; 搬送_戻り位置_GO_OFF
AND 201.11  ; 搬送_戻り位置_GO_ON
OUT 201.12  ; 搬送_戻り位置_GO_OFF
; rung 13
@LD 1.07  ; RB:PEND_主軸
OR 201.13  ; 搬送_戻り位置_END
AND 201.12  ; 搬送_戻り位置_GO_OFF
OUT 201.13  ; 搬送_戻り位置_END
TIMH(015) 0209 #3
; rung 14
LD T0209
OUT 201.14  ; 搬送C/E_F
; rung 15: RBO
@LD 60.06  ; 主軸RB_Pos1_END
@OR 201.13  ; 搬送_戻り位置_END
@OR 204.03  ; M_Pos1_END
@LD 202.01  ; 搬送搬送_位置
OR 252.00  ; ER:主軸RB
KEEP(011) 202.00  ; 搬送戻り_位置

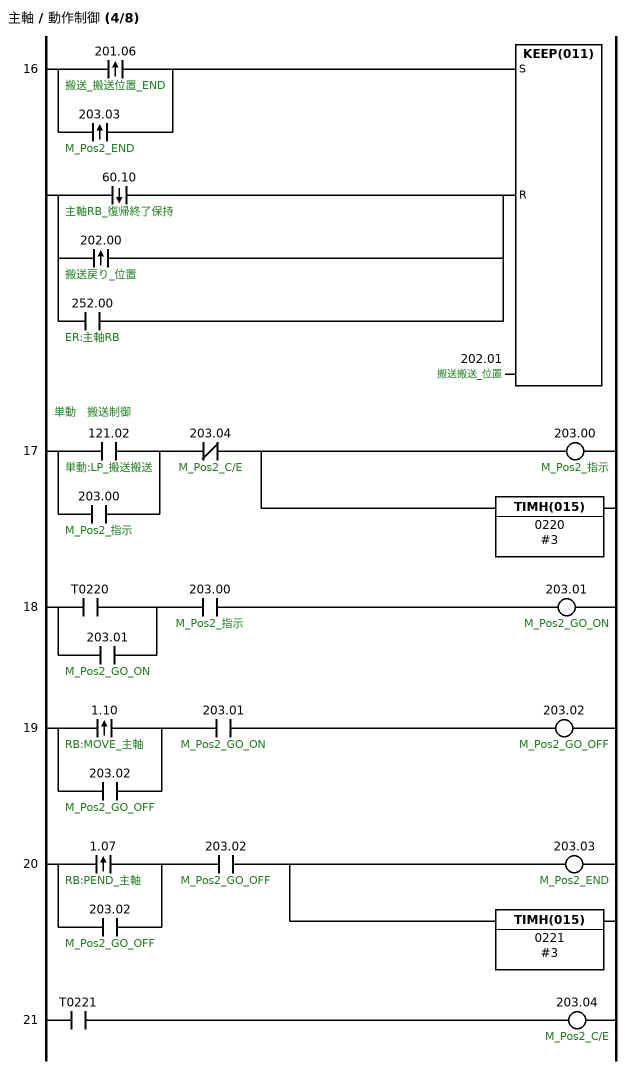
; rung 16
@LD 201.06  ; 搬送_搬送位置_END
@OR 203.03  ; M_Pos2_END
%LD 60.10  ; 主軸RB_復帰終了保持
@OR 202.00  ; 搬送戻り_位置
OR 252.00  ; ER:主軸RB
KEEP(011) 202.01  ; 搬送搬送_位置
; rung 17: 単動　搬送制御
LD 121.02  ; 単動:LP_搬送搬送
OR 203.00  ; M_Pos2_指示
ANDNOT 203.04  ; M_Pos2_C/E
OUT 203.00  ; M_Pos2_指示
TIMH(015) 0220 #3
; rung 18
LD T0220
OR 203.01  ; M_Pos2_GO_ON
AND 203.00  ; M_Pos2_指示
OUT 203.01  ; M_Pos2_GO_ON
; rung 19
@LD 1.10  ; RB:MOVE_主軸
OR 203.02  ; M_Pos2_GO_OFF
AND 203.01  ; M_Pos2_GO_ON
OUT 203.02  ; M_Pos2_GO_OFF
; rung 20
@LD 1.07  ; RB:PEND_主軸
OR 203.02  ; M_Pos2_GO_OFF
AND 203.02  ; M_Pos2_GO_OFF
OUT 203.03  ; M_Pos2_END
TIMH(015) 0221 #3
; rung 21
LD T0221
OUT 203.04  ; M_Pos2_C/E

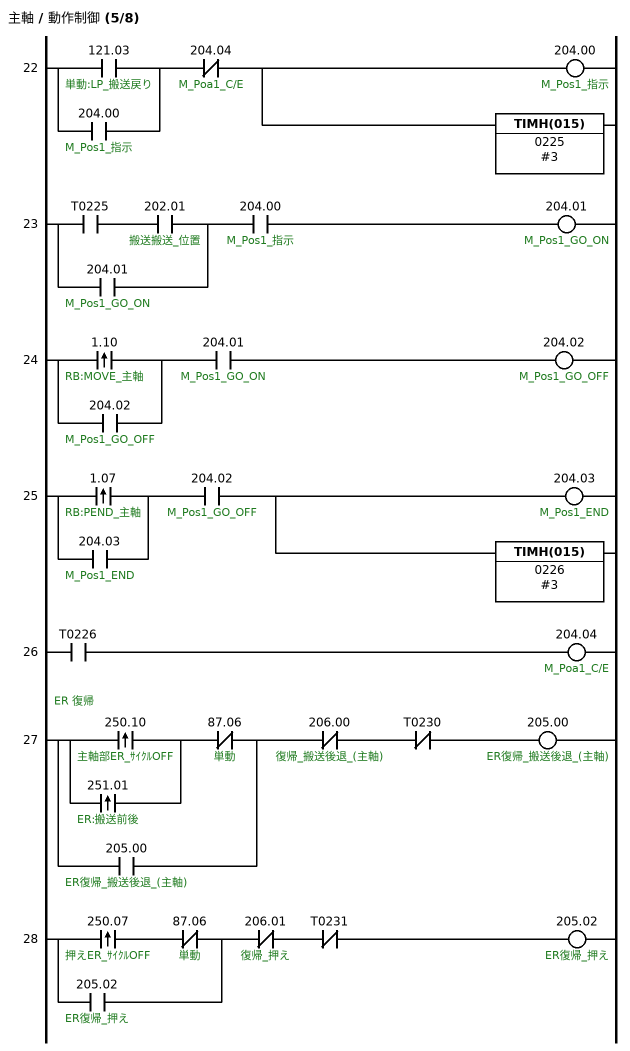
; rung 22
LD 121.03  ; 単動:LP_搬送戻り
OR 204.00  ; M_Pos1_指示
ANDNOT 204.04  ; M_Poa1_C/E
OUT 204.00  ; M_Pos1_指示
TIMH(015) 0225 #3
; rung 23
LD T0225
AND 202.01  ; 搬送搬送_位置
OR 204.01  ; M_Pos1_GO_ON
AND 204.00  ; M_Pos1_指示
OUT 204.01  ; M_Pos1_GO_ON
; rung 24
@LD 1.10  ; RB:MOVE_主軸
OR 204.02  ; M_Pos1_GO_OFF
AND 204.01  ; M_Pos1_GO_ON
OUT 204.02  ; M_Pos1_GO_OFF
; rung 25
@LD 1.07  ; RB:PEND_主軸
OR 204.03  ; M_Pos1_END
AND 204.02  ; M_Pos1_GO_OFF
OUT 204.03  ; M_Pos1_END
TIMH(015) 0226 #3
; rung 26
LD T0226
OUT 204.04  ; M_Poa1_C/E
; rung 27: ER 復帰
@LD 250.10  ; 主軸部ER_ｻｲｸﾙOFF
@OR 251.01  ; ER:搬送前後
ANDNOT 87.06  ; 単動
OR 205.00  ; ER復帰_搬送後退_(主軸)
ANDNOT 206.00  ; 復帰_搬送後退_(主軸)
ANDNOT T0230
OUT 205.00  ; ER復帰_搬送後退_(主軸)
; rung 28
@LD 250.07  ; 押えER_ｻｲｸﾙOFF
ANDNOT 87.06  ; 単動
OR 205.02  ; ER復帰_押え
ANDNOT 206.01  ; 復帰_押え
ANDNOT T0231
OUT 205.02  ; ER復帰_押え

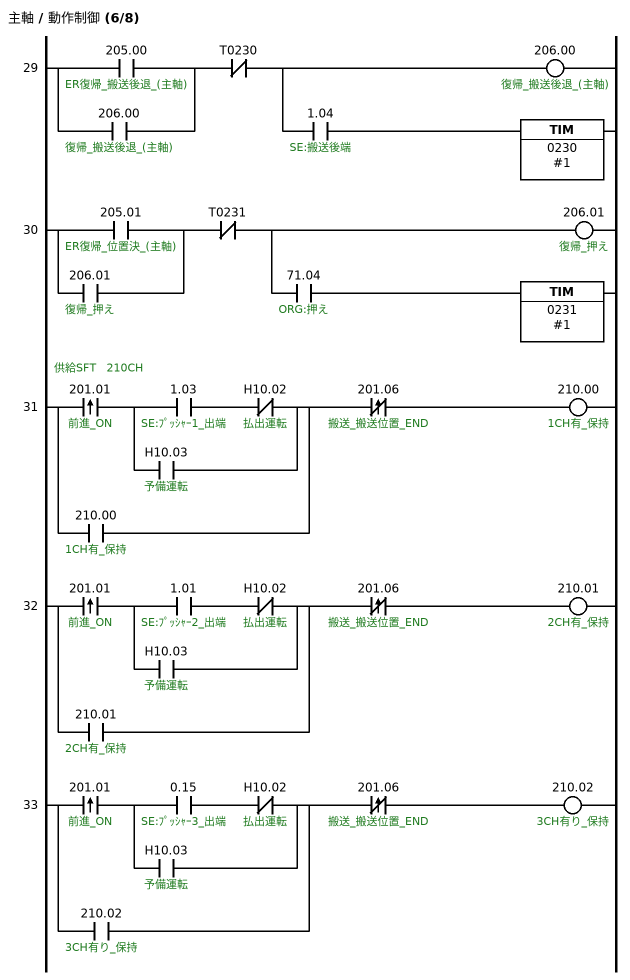
; rung 29
LD 205.00  ; ER復帰_搬送後退_(主軸)
OR 206.00  ; 復帰_搬送後退_(主軸)
ANDNOT T0230
OUT 206.00  ; 復帰_搬送後退_(主軸)
AND 1.04  ; SE:搬送後端
TIM 0230 #1
; rung 30
LD 205.01  ; ER復帰_位置決_(主軸)
OR 206.01  ; 復帰_押え
ANDNOT T0231
OUT 206.01  ; 復帰_押え
AND 71.04  ; ORG:押え
TIM 0231 #1
; rung 31: 供給SFT   210CH
@LD 201.01  ; 前進_ON
LD 1.03  ; SE:ﾌﾟｯｼｬｰ1_出端
ANDNOT H10.02  ; 払出運転
OR H10.03  ; 予備運転
ANDLD
OR 210.00  ; 1CH有_保持
@ANDNOT 201.06  ; 搬送_搬送位置_END
OUT 210.00  ; 1CH有_保持
; rung 32
@LD 201.01  ; 前進_ON
LD 1.01  ; SE:ﾌﾟｯｼｬｰ2_出端
ANDNOT H10.02  ; 払出運転
OR H10.03  ; 予備運転
ANDLD
OR 210.01  ; 2CH有_保持
@ANDNOT 201.06  ; 搬送_搬送位置_END
OUT 210.01  ; 2CH有_保持
; rung 33
@LD 201.01  ; 前進_ON
LD 0.15  ; SE:ﾌﾟｯｼｬｰ3_出端
ANDNOT H10.02  ; 払出運転
OR H10.03  ; 予備運転
ANDLD
OR 210.02  ; 3CH有り_保持
@ANDNOT 201.06  ; 搬送_搬送位置_END
OUT 210.02  ; 3CH有り_保持

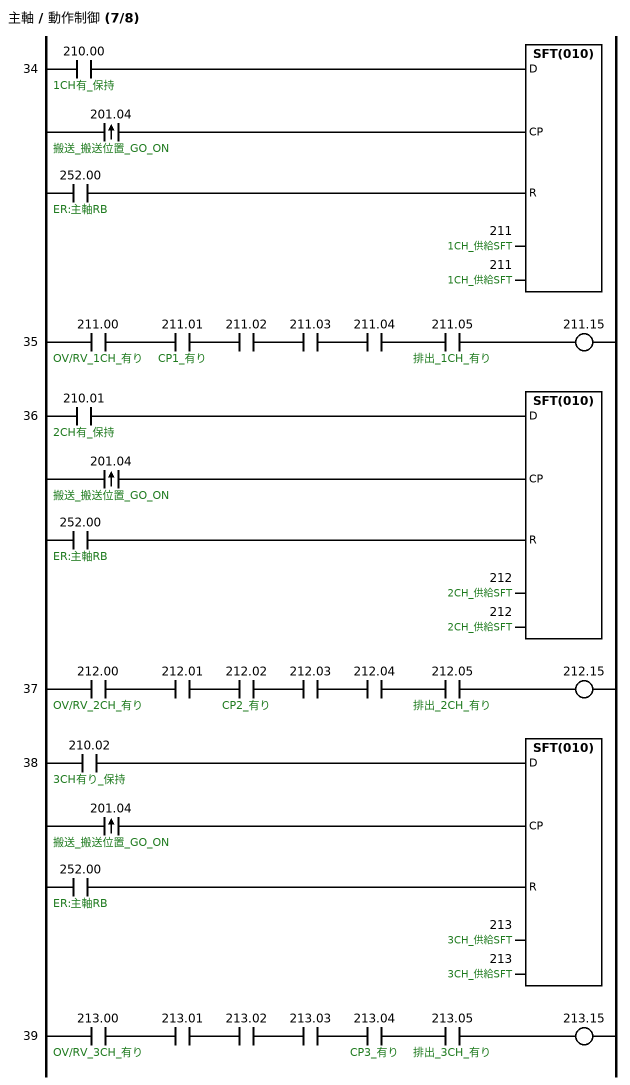
; rung 34
LD 210.00  ; 1CH有_保持
@LD 201.04  ; 搬送_搬送位置_GO_ON
LD 252.00  ; ER:主軸RB
SFT(010) 211 211  ; 1CH_供給SFT
; rung 35
LD 211.00  ; OV/RV_1CH_有り
AND 211.01  ; CP1_有り
AND 211.02
AND 211.03
AND 211.04
AND 211.05  ; 排出_1CH_有り
OUT 211.15
; rung 36
LD 210.01  ; 2CH有_保持
@LD 201.04  ; 搬送_搬送位置_GO_ON
LD 252.00  ; ER:主軸RB
SFT(010) 212 212  ; 2CH_供給SFT
; rung 37
LD 212.00  ; OV/RV_2CH_有り
AND 212.01
AND 212.02  ; CP2_有り
AND 212.03
AND 212.04
AND 212.05  ; 排出_2CH_有り
OUT 212.15
; rung 38
LD 210.02  ; 3CH有り_保持
@LD 201.04  ; 搬送_搬送位置_GO_ON
LD 252.00  ; ER:主軸RB
SFT(010) 213 213  ; 3CH_供給SFT
; rung 39
LD 213.00  ; OV/RV_3CH_有り
AND 213.01
AND 213.02
AND 213.03
AND 213.04  ; CP3_有り
AND 213.05  ; 排出_3CH_有り
OUT 213.15

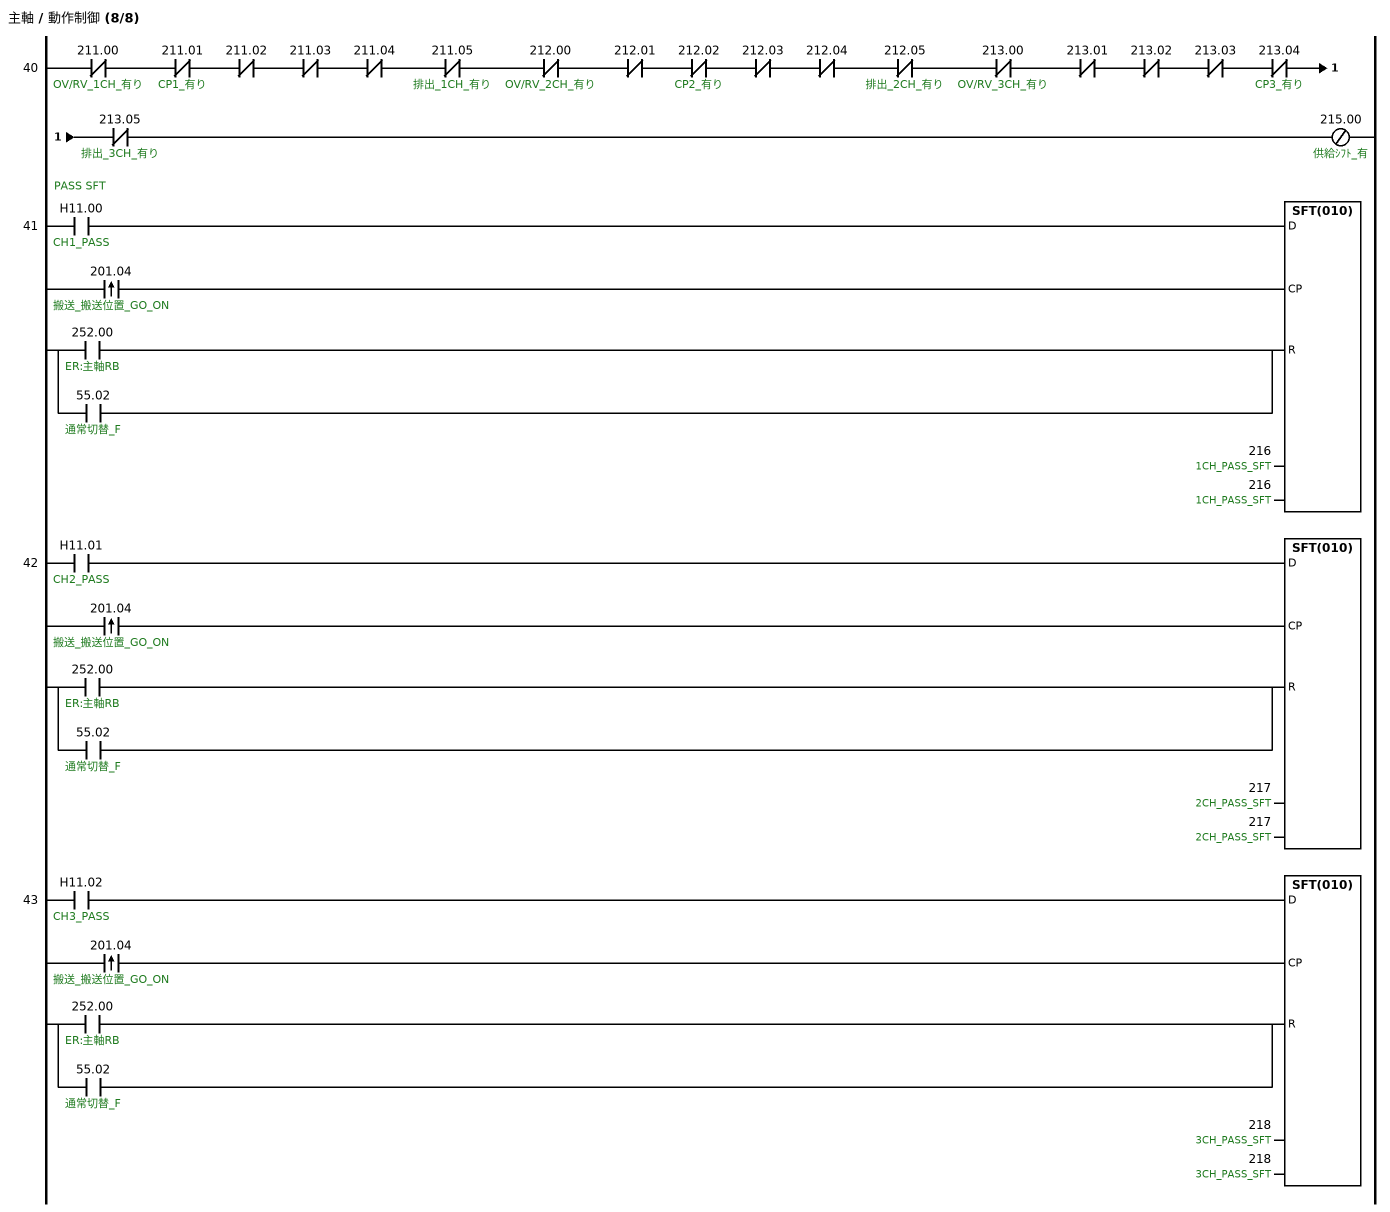
; rung 40
LDNOT 211.00  ; OV/RV_1CH_有り
ANDNOT 211.01  ; CP1_有り
ANDNOT 211.02
ANDNOT 211.03
ANDNOT 211.04
ANDNOT 211.05  ; 排出_1CH_有り
ANDNOT 212.00  ; OV/RV_2CH_有り
ANDNOT 212.01
ANDNOT 212.02  ; CP2_有り
ANDNOT 212.03
ANDNOT 212.04
ANDNOT 212.05  ; 排出_2CH_有り
ANDNOT 213.00  ; OV/RV_3CH_有り
ANDNOT 213.01
ANDNOT 213.02
ANDNOT 213.03
ANDNOT 213.04  ; CP3_有り
ANDNOT 213.05  ; 排出_3CH_有り
OUTNOT 215.00  ; 供給ｼﾌﾄ_有
; rung 41: PASS SFT
LD H11.00  ; CH1_PASS
@LD 201.04  ; 搬送_搬送位置_GO_ON
LD 252.00  ; ER:主軸RB
OR 55.02  ; 通常切替_F
SFT(010) 216 216  ; 1CH_PASS_SFT
; rung 42
LD H11.01  ; CH2_PASS
@LD 201.04  ; 搬送_搬送位置_GO_ON
LD 252.00  ; ER:主軸RB
OR 55.02  ; 通常切替_F
SFT(010) 217 217  ; 2CH_PASS_SFT
; rung 43
LD H11.02  ; CH3_PASS
@LD 201.04  ; 搬送_搬送位置_GO_ON
LD 252.00  ; ER:主軸RB
OR 55.02  ; 通常切替_F
SFT(010) 218 218  ; 3CH_PASS_SFT

### Section 出力

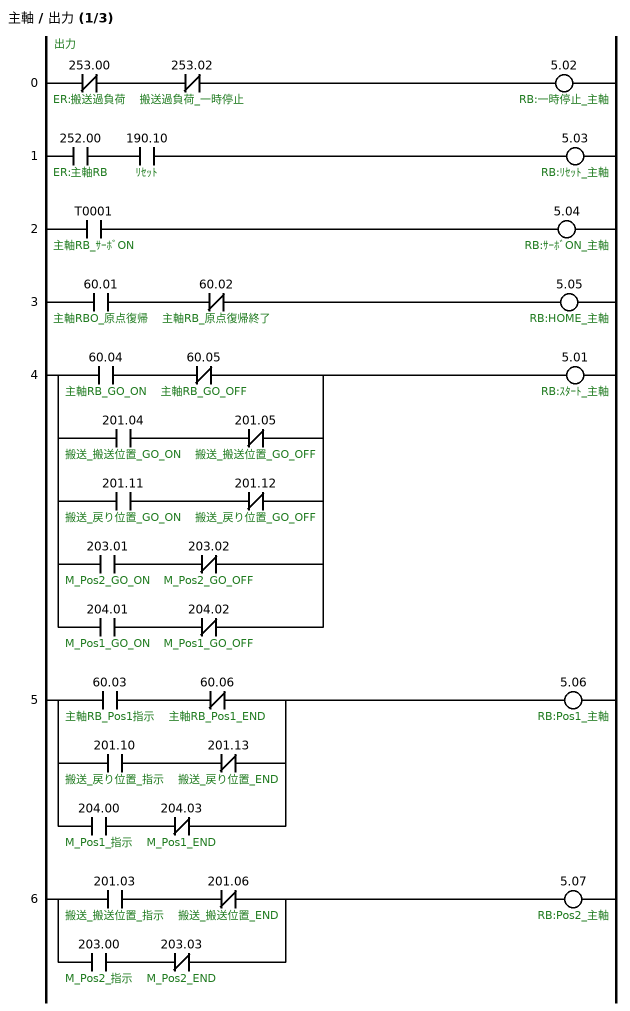
; rung 0: 出力
LDNOT 253.00  ; ER:搬送過負荷
ANDNOT 253.02  ; 搬送過負荷_一時停止
OUT 5.02  ; RB:一時停止_主軸
; rung 1
LD 252.00  ; ER:主軸RB
AND 190.10  ; ﾘｾｯﾄ
OUT 5.03  ; RB:ﾘｾｯﾄ_主軸
; rung 2
LD T0001  ; 主軸RB_ｻｰﾎﾞON
OUT 5.04  ; RB:ｻｰﾎﾞON_主軸
; rung 3
LD 60.01  ; 主軸RBO_原点復帰
ANDNOT 60.02  ; 主軸RB_原点復帰終了
OUT 5.05  ; RB:HOME_主軸
; rung 4
LD 60.04  ; 主軸RB_GO_ON
ANDNOT 60.05  ; 主軸RB_GO_OFF
LD 201.04  ; 搬送_搬送位置_GO_ON
ANDNOT 201.05  ; 搬送_搬送位置_GO_OFF
ORLD
LD 201.11  ; 搬送_戻り位置_GO_ON
ANDNOT 201.12  ; 搬送_戻り位置_GO_OFF
ORLD
LD 203.01  ; M_Pos2_GO_ON
ANDNOT 203.02  ; M_Pos2_GO_OFF
ORLD
LD 204.01  ; M_Pos1_GO_ON
ANDNOT 204.02  ; M_Pos1_GO_OFF
ORLD
OUT 5.01  ; RB:ｽﾀｰﾄ_主軸
; rung 5
LD 60.03  ; 主軸RB_Pos1指示
ANDNOT 60.06  ; 主軸RB_Pos1_END
LD 201.10  ; 搬送_戻り位置_指示
ANDNOT 201.13  ; 搬送_戻り位置_END
ORLD
LD 204.00  ; M_Pos1_指示
ANDNOT 204.03  ; M_Pos1_END
ORLD
OUT 5.06  ; RB:Pos1_主軸
; rung 6
LD 201.03  ; 搬送_搬送位置_指示
ANDNOT 201.06  ; 搬送_搬送位置_END
LD 203.00  ; M_Pos2_指示
ANDNOT 203.03  ; M_Pos2_END
ORLD
OUT 5.07  ; RB:Pos2_主軸

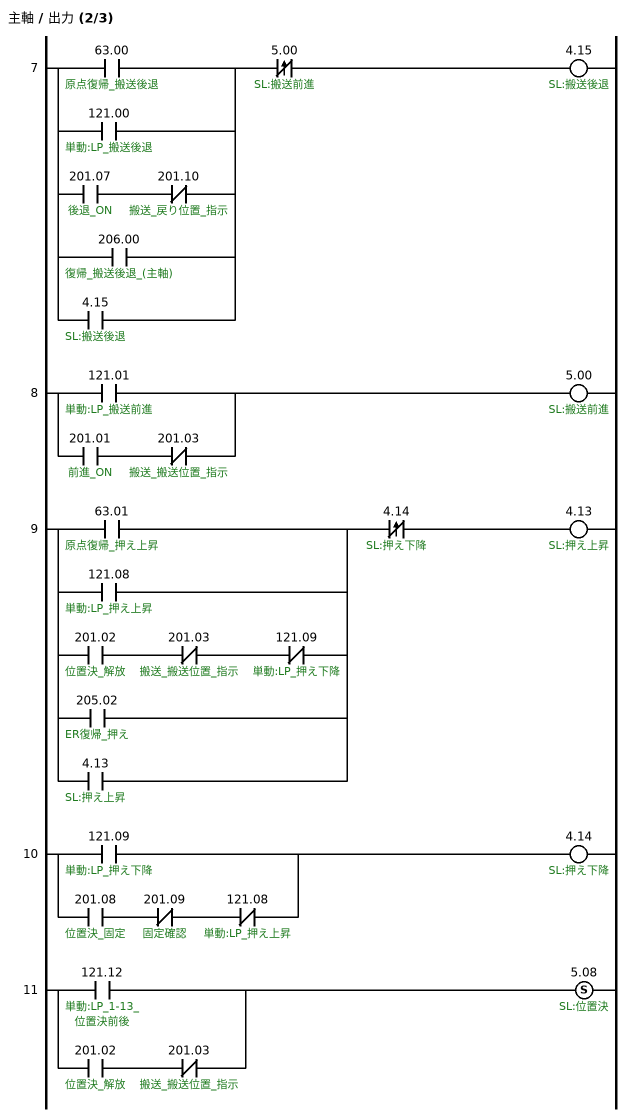
; rung 7
LD 63.00  ; 原点復帰_搬送後退
OR 121.00  ; 単動:LP_搬送後退
LD 201.07  ; 後退_ON
ANDNOT 201.10  ; 搬送_戻り位置_指示
ORLD
OR 206.00  ; 復帰_搬送後退_(主軸)
OR 4.15  ; SL:搬送後退
@ANDNOT 5.00  ; SL:搬送前進
OUT 4.15  ; SL:搬送後退
; rung 8
LD 121.01  ; 単動:LP_搬送前進
LD 201.01  ; 前進_ON
ANDNOT 201.03  ; 搬送_搬送位置_指示
ORLD
OUT 5.00  ; SL:搬送前進
; rung 9
LD 63.01  ; 原点復帰_押え上昇
OR 121.08  ; 単動:LP_押え上昇
LD 201.02  ; 位置決_解放
ANDNOT 201.03  ; 搬送_搬送位置_指示
ANDNOT 121.09  ; 単動:LP_押え下降
ORLD
OR 205.02  ; ER復帰_押え
OR 4.13  ; SL:押え上昇
@ANDNOT 4.14  ; SL:押え下降
OUT 4.13  ; SL:押え上昇
; rung 10
LD 121.09  ; 単動:LP_押え下降
LD 201.08  ; 位置決_固定
ANDNOT 201.09  ; 固定確認
ANDNOT 121.08  ; 単動:LP_押え上昇
ORLD
OUT 4.14  ; SL:押え下降
; rung 11
LD 121.12  ; 単動:LP_1-13_位置決前後
LD 201.02  ; 位置決_解放
ANDNOT 201.03  ; 搬送_搬送位置_指示
ORLD
SET 5.08  ; SL:位置決

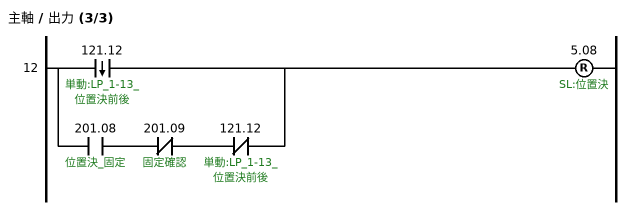
; rung 12
%LD 121.12  ; 単動:LP_1-13_位置決前後
LD 201.08  ; 位置決_固定
ANDNOT 201.09  ; 固定確認
ANDNOT 121.12  ; 単動:LP_1-13_位置決前後
ORLD
RSET 5.08  ; SL:位置決

### Section ｴﾗｰ

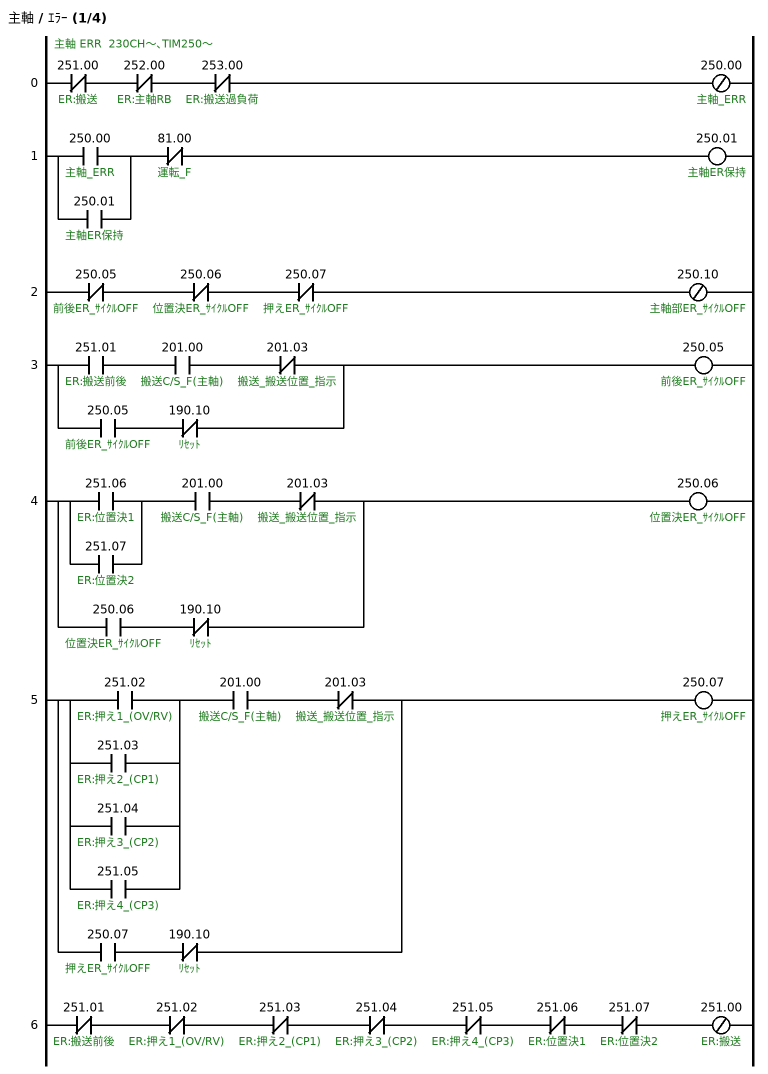
; rung 0: 主軸 ERR  230CH～､TIM250～
LDNOT 251.00  ; ER:搬送
ANDNOT 252.00  ; ER:主軸RB
ANDNOT 253.00  ; ER:搬送過負荷
OUTNOT 250.00  ; 主軸_ERR
; rung 1
LD 250.00  ; 主軸_ERR
OR 250.01  ; 主軸ER保持
ANDNOT 81.00  ; 運転_F
OUT 250.01  ; 主軸ER保持
; rung 2
LDNOT 250.05  ; 前後ER_ｻｲｸﾙOFF
ANDNOT 250.06  ; 位置決ER_ｻｲｸﾙOFF
ANDNOT 250.07  ; 押えER_ｻｲｸﾙOFF
OUTNOT 250.10  ; 主軸部ER_ｻｲｸﾙOFF
; rung 3
LD 251.01  ; ER:搬送前後
AND 201.00  ; 搬送C/S_F(主軸)
ANDNOT 201.03  ; 搬送_搬送位置_指示
LD 250.05  ; 前後ER_ｻｲｸﾙOFF
ANDNOT 190.10  ; ﾘｾｯﾄ
ORLD
OUT 250.05  ; 前後ER_ｻｲｸﾙOFF
; rung 4
LD 251.06  ; ER:位置決1
OR 251.07  ; ER:位置決2
AND 201.00  ; 搬送C/S_F(主軸)
ANDNOT 201.03  ; 搬送_搬送位置_指示
LD 250.06  ; 位置決ER_ｻｲｸﾙOFF
ANDNOT 190.10  ; ﾘｾｯﾄ
ORLD
OUT 250.06  ; 位置決ER_ｻｲｸﾙOFF
; rung 5
LD 251.02  ; ER:押え1_(OV/RV)
OR 251.03  ; ER:押え2_(CP1)
OR 251.04  ; ER:押え3_(CP2)
OR 251.05  ; ER:押え4_(CP3)
AND 201.00  ; 搬送C/S_F(主軸)
ANDNOT 201.03  ; 搬送_搬送位置_指示
LD 250.07  ; 押えER_ｻｲｸﾙOFF
ANDNOT 190.10  ; ﾘｾｯﾄ
ORLD
OUT 250.07  ; 押えER_ｻｲｸﾙOFF
; rung 6
LDNOT 251.01  ; ER:搬送前後
ANDNOT 251.02  ; ER:押え1_(OV/RV)
ANDNOT 251.03  ; ER:押え2_(CP1)
ANDNOT 251.04  ; ER:押え3_(CP2)
ANDNOT 251.05  ; ER:押え4_(CP3)
ANDNOT 251.06  ; ER:位置決1
ANDNOT 251.07  ; ER:位置決2
OUTNOT 251.00  ; ER:搬送

